// TIA Portal V18 export
DATA_BLOCK "HeatingPLC_vDI_Vars"   // DB11003
{ S7_Optimized_Access := 'FALSE' }
VERSION : 0.1
// stored: AutoNumber false, DBAccessibleFromOPCUA true, IsOnlyStoredInLoadMemory false, IsWriteProtectedInAS false
   VAR
      vDI1 { S7_SetPoint := 'True'} : "UDT_vDI";
      vDI2 { S7_SetPoint := 'True'} : "UDT_vDI";
      vDI3 { S7_SetPoint := 'True'} : "UDT_vDI";
      vDI4 { S7_SetPoint := 'True'} : "UDT_vDI";
      vDI5 { S7_SetPoint := 'True'} : "UDT_vDI";
      vDI6 { S7_SetPoint := 'True'} : "UDT_vDI";
      vDI7 { S7_SetPoint := 'True'} : "UDT_vDI";
      vDI8 { S7_SetPoint := 'True'} : "UDT_vDI";
   END_VAR
BEGIN
END_DATA_BLOCK
